FUNCTION_BLOCK Test_TStringSplitter_Handles_Empty_SubString EXTENDS T_UnitTestBase
VAR
    StringSplitter : T_StringSplitter;
    SubjectString  : T_MaxString := 'Badger,';
END_VAR

{attribute 'analysis' := '-33'} // inhibit unused variable warning
METHOD RunTest
IF Retest THEN
	SUPER^.Init();
END_IF

IF TestCompleted THEN
	RETURN;
END_IF

StringSplitter.Init(Str    := SubjectString,
                    Delim1 := ',',
                    Delim2 := '');

AssertEquals_STRING(Expected := 'Badger',
                    Actual   := StringSplitter.GetNext(),
                    Message  := 'StringSplitter.GetNext()');

AssertEquals_BOOL(Expected := FALSE,
                  Actual   := StringSplitter.HasMore(),
                  Message  := 'StringSplitter.HasMore()');

AssertEquals_STRING(Expected := '',
                    Actual   := StringSplitter.GetNext(),
                    Message  := 'StringSplitter.GetNext()');

TestCompleted := TRUE;
END_METHOD

END_FUNCTION_BLOCK

(* stored: Version 1.1.0.1, ProductVersion 3.1.4024.12
   POU Test_TStringSplitter_Handles_Empty_SubString: Id {b7ce1263-3bd7-0eb9-2316-2cc2cba02503}, SpecialFunc None
   Method RunTest: Id {22d44373-85be-060a-375b-6299242a53f7} *)
